{attribute 'OPC.UA.DA.JobMethod' := 'JobMethode_SecuringProcess'}
FUNCTION_BLOCK MBS_MR01_AS_SecuringProcess
VAR
	AlwaysTrue : BOOL := TRUE;
	// Used for debugging purposes to display InputArguments of method call
	MethodCall_SecuringProcess : BOOL := FALSE; // used to store InputArg "MethodCall" from Start() method
	ResetMethodCall	: BOOL := FALSE;	
	SecuringTime : TIME;	//Time for Securing the Workpiece
	SecuringProcessingTime : TIME; //Two Times for Securing the Workpiece (for Secure and Release) + HardeningProcessingTime
	callCounterStart : ULINT; // counts how many times the Start() method has been called
	callCounterCheckState : ULINT; // counts how many times the CheckState() method has been called
	callCounterAbort : ULINT; // counts how many times the Abort() method has been called
	
	// Variables to determine if a job has been started (Start() method has been called) or finished
	jobRunning : BOOL;
	jobFinished : BOOL;

	// State machine variable
	state : UDINT;
	
	//Variablen des FBs
	MBS_MR01_SecuringProcess : SecuringWorkpiece;
END_VAR
	
VAR_INPUT
	ESS: BOOL;
	TouchSensor_01 : BOOL;
	AutomaticMode: BOOL;
END_VAR

VAR_OUTPUT
	DO_SecuringProcessCompressorMR01_01 : BOOL;
	DO_SecuringProcessValveMR01_02 : BOOL;
END_VAR

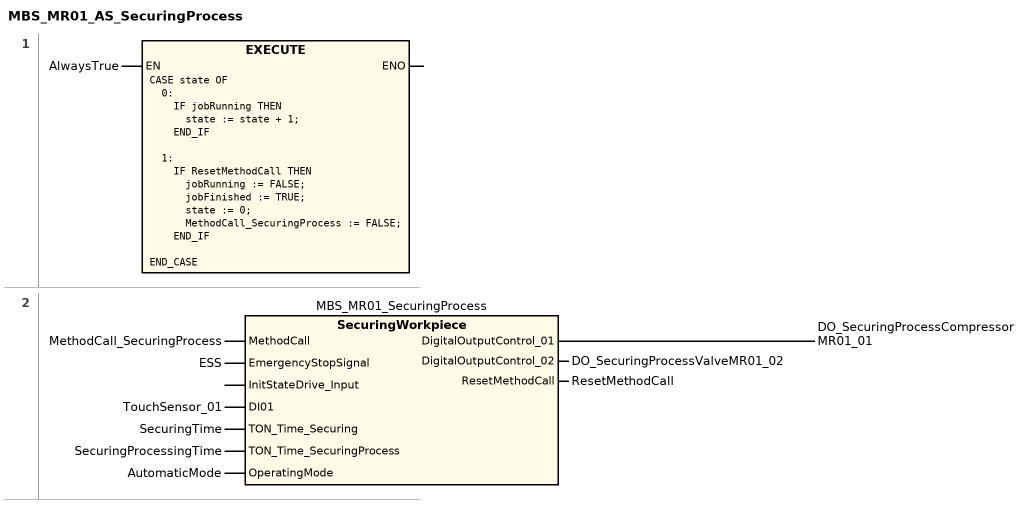
// NETWORK 1
IF AlwaysTrue THEN
    CASE state OF
    	0:
    		IF jobRunning THEN
    			state := state + 1;
    		END_IF
    		
    	1:
    		IF ResetMethodCall THEN
    			jobRunning := FALSE;
    			jobFinished := TRUE;
    			state := 0;
    			MethodCall_SecuringProcess := FALSE;
    		END_IF
    		
    END_CASE
END_IF

// NETWORK 2
MBS_MR01_SecuringProcess(
    MethodCall := MethodCall_SecuringProcess,
    EmergencyStopSignal := ESS,
    DI01 := TouchSensor_01,
    TON_Time_Securing := SecuringTime,
    TON_Time_SecuringProcess := SecuringProcessingTime,
    OperatingMode := AutomaticMode,
    DigitalOutputControl_02 => DO_SecuringProcessValveMR01_02,
    ResetMethodCall => ResetMethodCall); // SecuringWorkpiece
DO_SecuringProcessCompressorMR01_01 := MBS_MR01_SecuringProcess.DigitalOutputControl_01;

{attribute 'TcRpcEnable' := '1'}
METHOD Abort : HRESULT
VAR_INPUT
	hdl : UDINT; // Do not change, used by server.
END_VAR
callCounterAbort := callCounterAbort + 1;
END_METHOD

{attribute 'TcRpcEnable' := '1'}
METHOD CheckState : HRESULT
VAR_INPUT
	hdl : UDINT; // Do not change, used by server.
END_VAR
VAR_OUTPUT
	bBusy : BOOL; // Do not change. Used by server to find out if the job is finished
	
	// List of OutputArguments for OPC UA method, may be customized
	State : BOOL; // Abgeschlossener MethodCall
	MethodCall: BOOL; //Input Recall
END_VAR
callCounterCheckState := callCounterCheckState + 1;
IF NOT jobFinished THEN
	bBusy := TRUE; // job is not finished yet
	CheckState := 0; // no error
ELSE
	bBusy := FALSE; // job is finished
	CheckState := 0; // done, no error occured during execution (OPC UA StatusCode "GOOD")
	jobFinished := FALSE;
	State := ResetMethodCall;
	MethodCall := MethodCall_SecuringProcess;
END_IF
END_METHOD

{attribute 'TcRpcEnable' := '1'}
METHOD Start : HRESULT
VAR_INPUT
	// List of InputArguments for OPC UA method, may be customized
	MethodCall : BOOL; // some description
	Securing_Time : TIME;
	SecuringProcessing_Time : TIME;
END_VAR
VAR_OUTPUT
	hdl : UDINT; // Do not change, used by server.
END_VAR
callCounterStart := callCounterStart + 1;

MethodCall_SecuringProcess := MethodCall;
SecuringTime := Securing_Time;
SecuringProcessingTime := SecuringProcessing_Time;

jobRunning := TRUE;
Start := 0; // no error occured, e.g. while parsing the input arguments (0 = OPC UA StatusCode "GOOD")
END_METHOD

END_FUNCTION_BLOCK

(* stored: Version 1.1.0.1, ProductVersion 3.1.4026.18
   POU MBS_MR01_AS_SecuringProcess: Id {2b1534eb-d527-431b-9fb5-33274cbac8f1}, SpecialFunc None
   Method Abort: Id {0da98f48-656c-4805-89ab-798246fcb813}
   Method CheckState: Id {d74b50de-72c0-484f-b3a6-e7c7388e8f18}
   Method Start: Id {4a4d1364-afb9-4324-a632-f637c79ad412} *)
